FUNCTION_BLOCK Central_Server (* Blake Central Server *)
  (* Standard: 61499-2 *)
  (* Version 0.2, 2003-12-04, JHC, Rockwell Automation, Renamed for better indexing. *)
  (* Version 0.1, 2002-11-05, JHC, Rockwell Automation, Corrected missing ST element in Algorithm REQ. *)
  (* Version 0.0, 2000-05-30, JHC, Rockwell Automation *)
  (* Compiler header: package fb.rt.cs725; *)
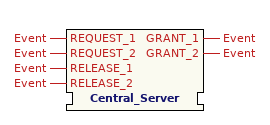
  EVENT_INPUT
    REQUEST_1;
    REQUEST_2;
    RELEASE_1;
    RELEASE_2;
  END_EVENT
  EVENT_OUTPUT
    GRANT_1;
    GRANT_2;
  END_EVENT
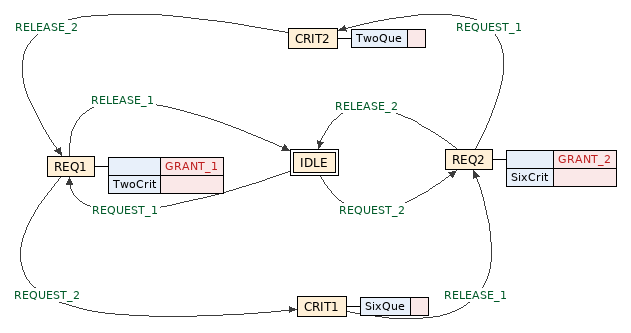
  EC_STATES
    IDLE; (* INIT *)
    REQ2 : -> GRANT_2, SixCrit;
    REQ1 : -> GRANT_1, TwoCrit;
    CRIT2 : TwoQue;
    CRIT1 : SixQue;
  END_STATES
  EC_TRANSITIONS
    IDLE TO REQ2 := REQUEST_2;
    REQ2 TO IDLE := RELEASE_2;
    IDLE TO REQ1 := REQUEST_1;
    REQ1 TO IDLE := RELEASE_1;
    REQ2 TO CRIT2 := REQUEST_1;
    CRIT2 TO REQ1 := RELEASE_2;
    REQ1 TO CRIT1 := REQUEST_2;
    CRIT1 TO REQ2 := RELEASE_1;
  END_TRANSITIONS
  ALGORITHM TwoQue IN Java: (* Initialization algorithm *)
System.out.println("Converyor TWO in queue");
  END_ALGORITHM
  ALGORITHM TwoCrit IN Java: (* Initialization algorithm *)
System.out.println("Converyor Two accessing thecritical section");
  END_ALGORITHM
  ALGORITHM SixQue IN Java: (* Initialization algorithm *)
System.out.println("Converyor Six in queue");
  END_ALGORITHM
  ALGORITHM SixCrit IN Java: (* Initialization algorithm *)
System.out.println("Converyor Six accessing the critical section");
  END_ALGORITHM
END_FUNCTION_BLOCK
